# EPICS autosave request: andor3App/Db/andor3_settings.req
$(P)$(R)FrameRate
$(P)$(R)PreAmpGain
$(P)$(R)ReadoutRate
$(P)$(R)Overlap
$(P)$(R)NoiseFilter
$(P)$(R)PixelEncoding
$(P)$(R)A3Binning
$(P)$(R)A3ShutterMode
$(P)$(R)SensorCooling
$(P)$(R)TempControl
$(P)$(R)FanSpeed
$(P)$(R)GateMode
$(P)$(R)InsertionDelay
$(P)$(R)MCPIntelligate
$(P)$(R)MCPGain
$(P)$(R)DDGOutputDelay
$(P)$(R)DDGOutputEnable
$(P)$(R)DDGOutputPolarity
$(P)$(R)DDGOutputSelect
$(P)$(R)DDGOutputStepEnable
$(P)$(R)DDGOutputWidth
$(P)$(R)DDGStepEnabled
$(P)$(R)DDGStepDelayMode
$(P)$(R)DDGStepDelayCoefficientA
$(P)$(R)DDGStepDelayCoefficientB
$(P)$(R)DDGStepWidthMode
$(P)$(R)DDGStepWidthCoefficientA
$(P)$(R)DDGStepWidthCoefficientB
file "ADBase_settings.req", P=$(P), R=$(R)
